// TIA Portal V19 export
DATA_BLOCK "MobilePanel"   // DB1071
{ S7_Optimized_Access := 'FALSE' }
// stored: AutoNumber false
   VAR
      Koordinierung : Word;
      Schluessel : Bool;
      Drucktaster_K2_LED : Int;
      Drucktaster_K2_Push : Bool;
   END_VAR
BEGIN
END_DATA_BLOCK
